Staubli VAL3: JointFbkMsg.dtx

public Header header
  [0]
    num nMsgType
    num nCommType
    num nReplyCode
    num nData[12]
public Prefix prefix
  [0]
    num nLength
    num nData[4]
public JointFeedback jointFeedback
  [0]
    num nRobotId
    num nValidFields
    num nTime
    num nPositions[10]
    num nVelocities[10]
    num nAccelerations[10]
public Body body
  [0]
    num nData[132]
